TYPE Array2Byte :
UNION
	arrByte 		:ARRAY[0..1] OF BYTE;
	sValue			:INT; 
END_UNION
END_TYPE

(* stored: Version 1.1.0.1
   DUT Array2Byte: Id {da3cbaf8-bf16-4594-bb27-09d6813e687a} *)
